INTERFACE I_OffCommand

PROPERTY IsOff : Bool
GET
END_GET
END_PROPERTY

METHOD Off
END_METHOD

END_INTERFACE

(* stored: Version 1.1.0.1, ProductVersion 3.1.4024.11
   Itf I_OffCommand: Id {9598dbd2-5ce8-4ed8-a51c-94df587af3e7}
   Property IsOff: Id {c8a07c24-29f7-45d3-bb08-f511d7e9341c}
   Get Get: Id {0bab355d-90ae-4fc9-b2f2-3c26eaf1f0e1}
   Method Off: Id {264ef751-5b49-4856-b742-1f4bafaea6d7} *)
